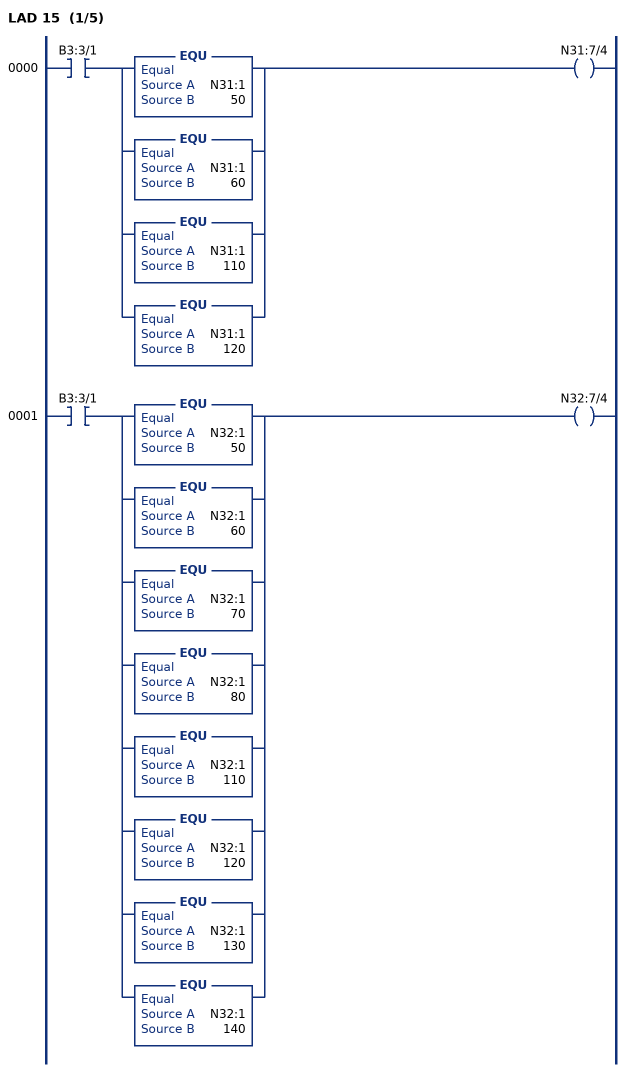
% Rung: 0 %
SOR XIC B3:3/1 BST EQU N31:1 50 NXB EQU N31:1 60 NXB EQU N31:1 110 NXB EQU N31:1 120 BND OTE N31:7/4 EOR
% Rung: 1 %
SOR XIC B3:3/1 BST EQU N32:1 50 NXB EQU N32:1 60 NXB EQU N32:1 70 NXB EQU N32:1 80 NXB EQU N32:1 110 NXB EQU N32:1 120 NXB EQU N32:1 130 NXB EQU N32:1 140 BND OTE N32:7/4 EOR

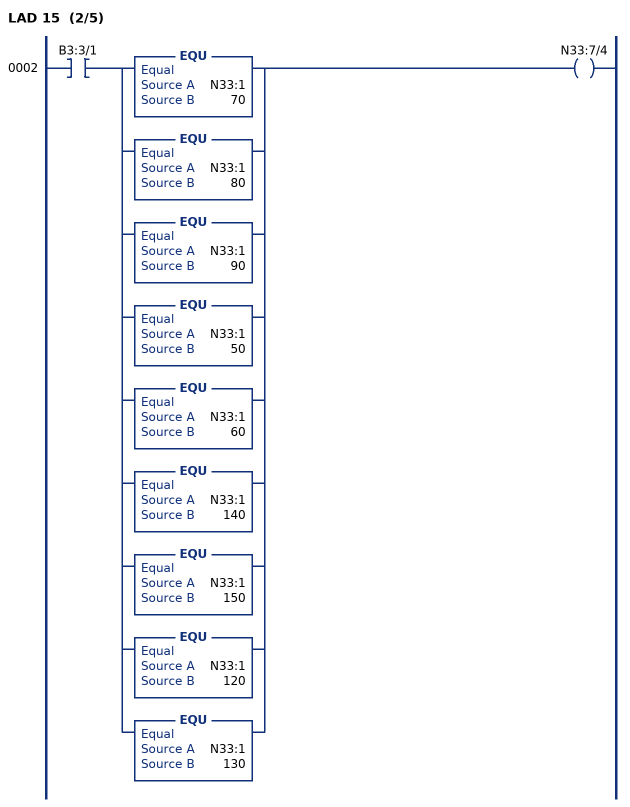
% Rung: 2 %
SOR XIC B3:3/1 BST EQU N33:1 70 NXB EQU N33:1 80 NXB EQU N33:1 90 NXB EQU N33:1 50 NXB EQU N33:1 60 NXB EQU N33:1 140 NXB EQU N33:1 150 NXB EQU N33:1 120 NXB EQU N33:1 130 BND OTE N33:7/4 EOR

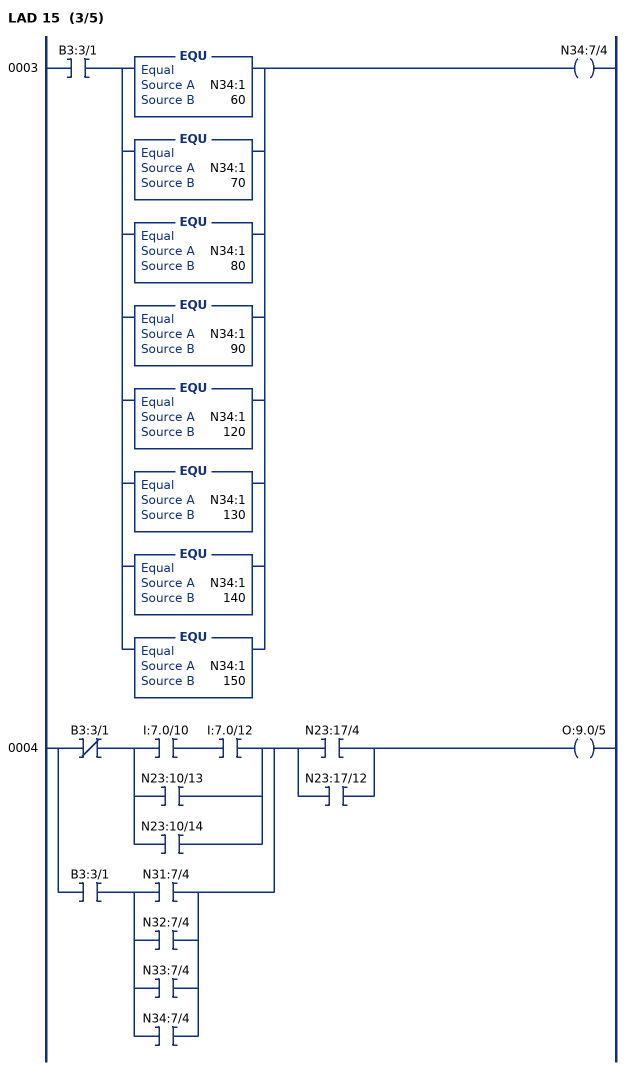
% Rung: 3 %
SOR XIC B3:3/1 BST EQU N34:1 60 NXB EQU N34:1 70 NXB EQU N34:1 80 NXB EQU N34:1 90 NXB EQU N34:1 120 NXB EQU N34:1 130 NXB EQU N34:1 140 NXB EQU N34:1 150 BND OTE N34:7/4 EOR
% Rung: 4 %
SOR BST XIO B3:3/1 BST XIC I:7.0/10 XIC I:7.0/12 NXB XIC N23:10/13 NXB XIC N23:10/14 BND NXB XIC B3:3/1 BST XIC N31:7/4 NXB XIC N32:7/4 NXB XIC N33:7/4 NXB XIC N34:7/4 BND BND BST XIC N23:17/4 NXB XIC N23:17/12 BND OTE O:9.0/5 EOR

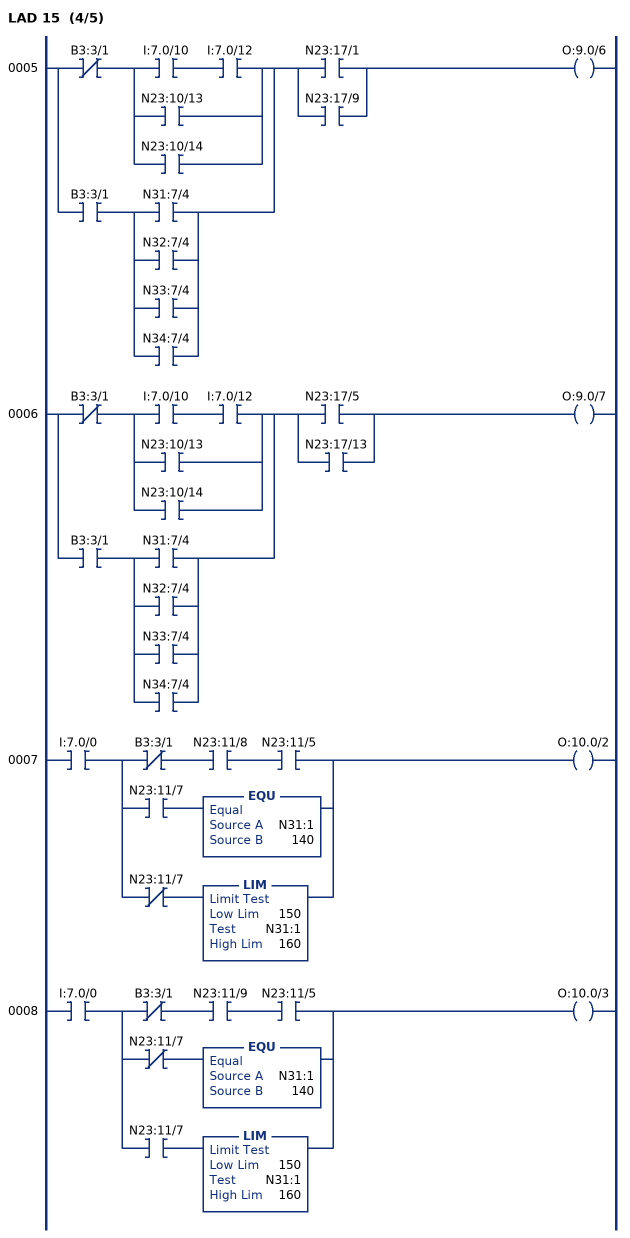
% Rung: 5 %
SOR BST XIO B3:3/1 BST XIC I:7.0/10 XIC I:7.0/12 NXB XIC N23:10/13 NXB XIC N23:10/14 BND NXB XIC B3:3/1 BST XIC N31:7/4 NXB XIC N32:7/4 NXB XIC N33:7/4 NXB XIC N34:7/4 BND BND BST XIC N23:17/1 NXB XIC N23:17/9 BND OTE O:9.0/6 EOR
% Rung: 6 %
SOR BST XIO B3:3/1 BST XIC I:7.0/10 XIC I:7.0/12 NXB XIC N23:10/13 NXB XIC N23:10/14 BND NXB XIC B3:3/1 BST XIC N31:7/4 NXB XIC N32:7/4 NXB XIC N33:7/4 NXB XIC N34:7/4 BND BND BST XIC N23:17/5 NXB XIC N23:17/13 BND OTE O:9.0/7 EOR
% Rung: 7 %
SOR XIC I:7.0/0 BST XIO B3:3/1 XIC N23:11/8 XIC N23:11/5 NXB XIC N23:11/7 EQU N31:1 140 NXB XIO N23:11/7 LIM 150 N31:1 160 BND OTE O:10.0/2 EOR
% Rung: 8 %
SOR XIC I:7.0/0 BST XIO B3:3/1 XIC N23:11/9 XIC N23:11/5 NXB XIO N23:11/7 EQU N31:1 140 NXB XIC N23:11/7 LIM 150 N31:1 160 BND OTE O:10.0/3 EOR

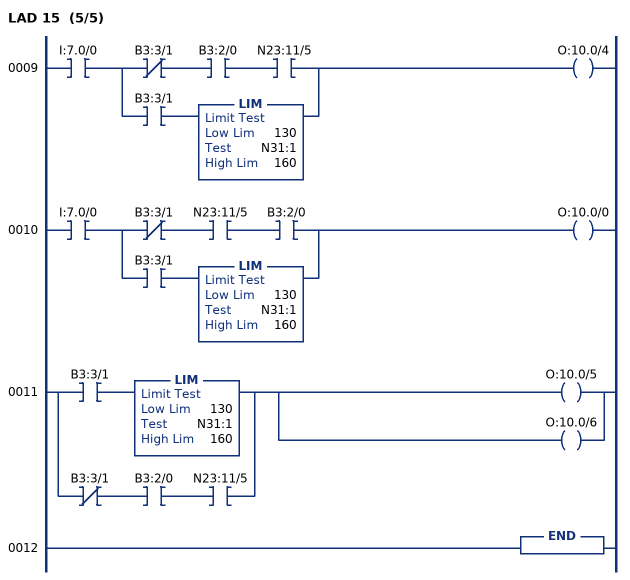
% Rung: 9 %
SOR XIC I:7.0/0 BST XIO B3:3/1 XIC B3:2/0 XIC N23:11/5 NXB XIC B3:3/1 LIM 130 N31:1 160 BND OTE O:10.0/4 EOR
% Rung: 10 %
SOR XIC I:7.0/0 BST XIO B3:3/1 XIC N23:11/5 XIC B3:2/0 NXB XIC B3:3/1 LIM 130 N31:1 160 BND OTE O:10.0/0 EOR
% Rung: 11 %
SOR BST XIC B3:3/1 LIM 130 N31:1 160 NXB XIO B3:3/1 XIC B3:2/0 XIC N23:11/5 BND BST OTE O:10.0/5 NXB OTE O:10.0/6 BND EOR
% Rung: 12 %
SOR END EOR

LADDER 21
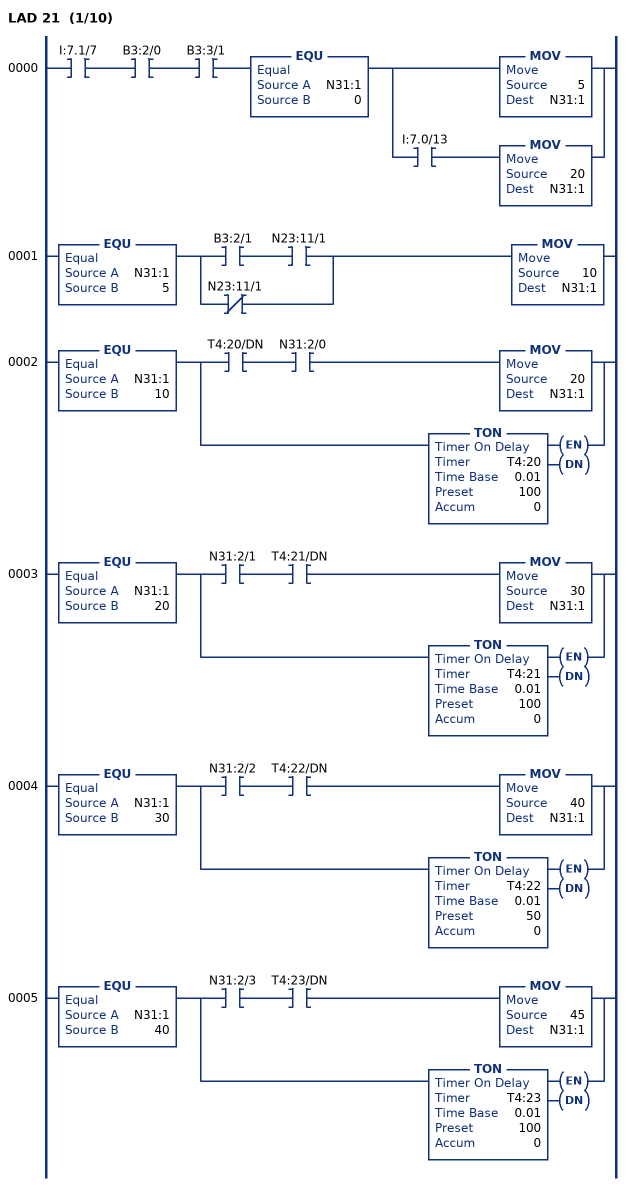
% Rung: 0 %
SOR XIC I:7.1/7 XIC B3:2/0 XIC B3:3/1 EQU N31:1 0 BST MOV 5 N31:1 NXB XIC I:7.0/13 MOV 20 N31:1 BND EOR
% Rung: 1 %
SOR EQU N31:1 5 BST XIC B3:2/1 XIC N23:11/1 NXB XIO N23:11/1 BND MOV 10 N31:1 EOR
% Rung: 2 %
SOR EQU N31:1 10 BST XIC T4:20/DN XIC N31:2/0 MOV 20 N31:1 NXB TON T4:20 0.01 100 0 BND EOR
% Rung: 3 %
SOR EQU N31:1 20 BST XIC N31:2/1 XIC T4:21/DN MOV 30 N31:1 NXB TON T4:21 0.01 100 0 BND EOR
% Rung: 4 %
SOR EQU N31:1 30 BST XIC N31:2/2 XIC T4:22/DN MOV 40 N31:1 NXB TON T4:22 0.01 50 0 BND EOR
% Rung: 5 %
SOR EQU N31:1 40 BST XIC N31:2/3 XIC T4:23/DN MOV 45 N31:1 NXB TON T4:23 0.01 100 0 BND EOR

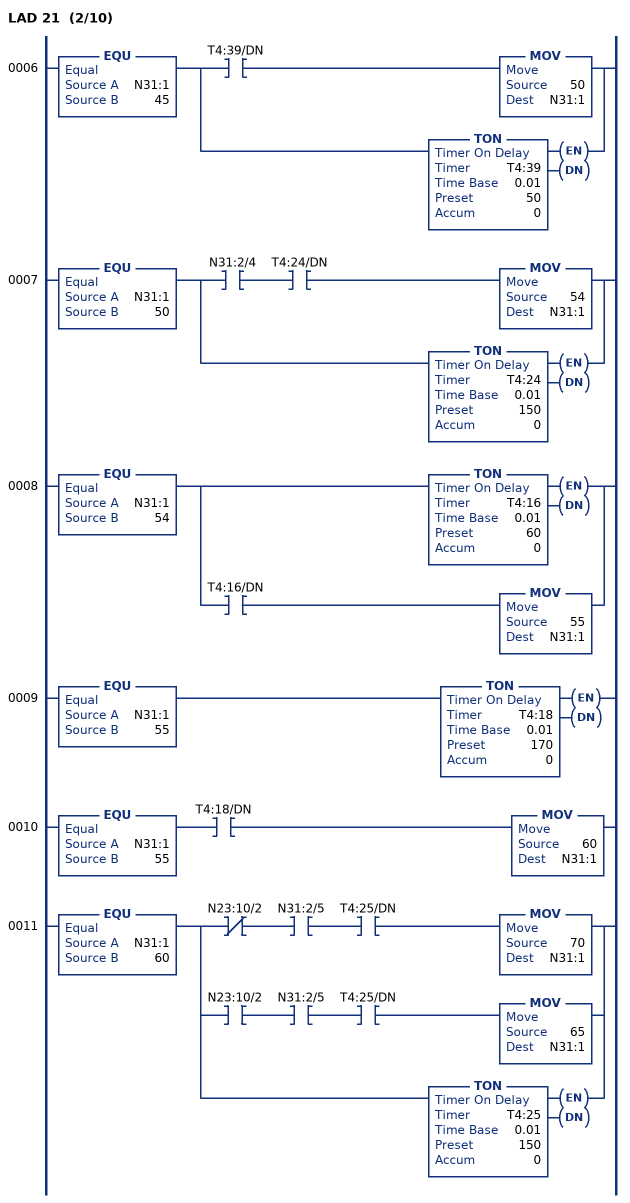
% Rung: 6 %
SOR EQU N31:1 45 BST XIC T4:39/DN MOV 50 N31:1 NXB TON T4:39 0.01 50 0 BND EOR
% Rung: 7 %
SOR EQU N31:1 50 BST XIC N31:2/4 XIC T4:24/DN MOV 54 N31:1 NXB TON T4:24 0.01 150 0 BND EOR
% Rung: 8 %
SOR EQU N31:1 54 BST TON T4:16 0.01 60 0 NXB XIC T4:16/DN MOV 55 N31:1 BND EOR
% Rung: 9 %
SOR EQU N31:1 55 TON T4:18 0.01 170 0 EOR
% Rung: 10 %
SOR EQU N31:1 55 XIC T4:18/DN MOV 60 N31:1 EOR
% Rung: 11 %
SOR EQU N31:1 60 BST XIO N23:10/2 XIC N31:2/5 XIC T4:25/DN MOV 70 N31:1 NXB XIC N23:10/2 XIC N31:2/5 XIC T4:25/DN MOV 65 N31:1 NXB TON T4:25 0.01 150 0 BND EOR

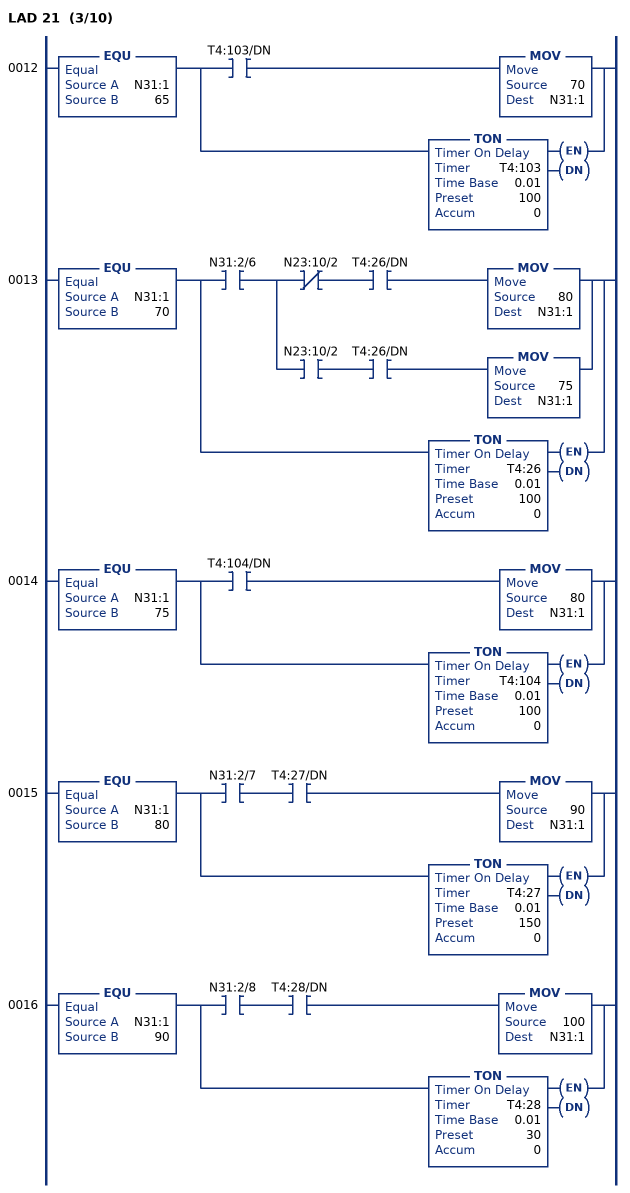
% Rung: 12 %
SOR EQU N31:1 65 BST XIC T4:103/DN MOV 70 N31:1 NXB TON T4:103 0.01 100 0 BND EOR
% Rung: 13 %
SOR EQU N31:1 70 BST XIC N31:2/6 BST XIO N23:10/2 XIC T4:26/DN MOV 80 N31:1 NXB XIC N23:10/2 XIC T4:26/DN MOV 75 N31:1 BND NXB TON T4:26 0.01 100 0 BND EOR
% Rung: 14 %
SOR EQU N31:1 75 BST XIC T4:104/DN MOV 80 N31:1 NXB TON T4:104 0.01 100 0 BND EOR
% Rung: 15 %
SOR EQU N31:1 80 BST XIC N31:2/7 XIC T4:27/DN MOV 90 N31:1 NXB TON T4:27 0.01 150 0 BND EOR
% Rung: 16 %
SOR EQU N31:1 90 BST XIC N31:2/8 XIC T4:28/DN MOV 100 N31:1 NXB TON T4:28 0.01 30 0 BND EOR

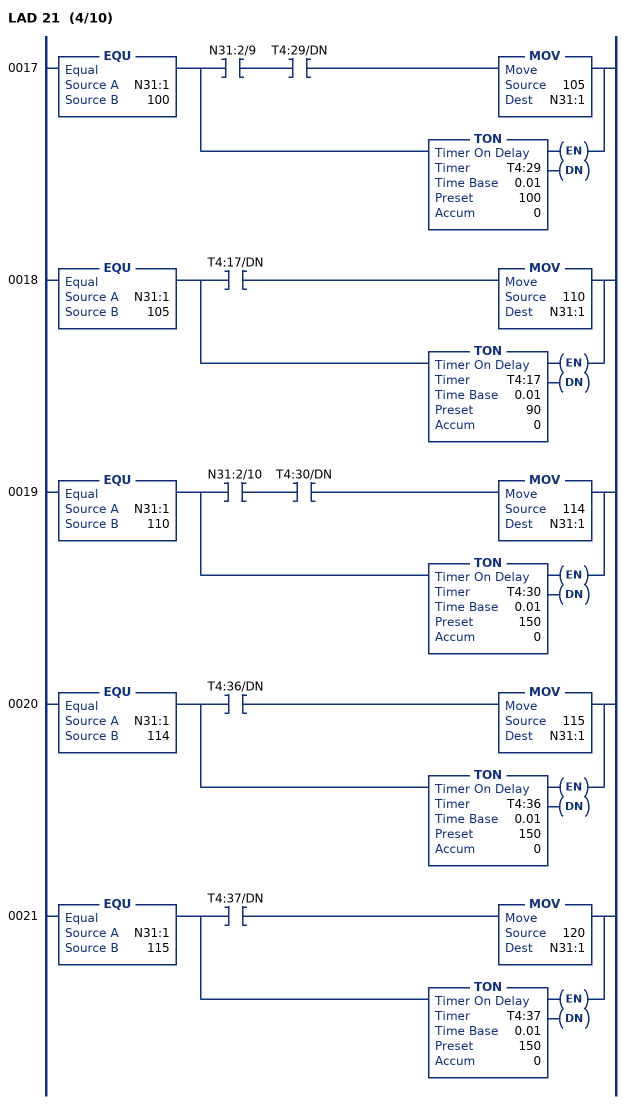
% Rung: 17 %
SOR EQU N31:1 100 BST XIC N31:2/9 XIC T4:29/DN MOV 105 N31:1 NXB TON T4:29 0.01 100 0 BND EOR
% Rung: 18 %
SOR EQU N31:1 105 BST XIC T4:17/DN MOV 110 N31:1 NXB TON T4:17 0.01 90 0 BND EOR
% Rung: 19 %
SOR EQU N31:1 110 BST XIC N31:2/10 XIC T4:30/DN MOV 114 N31:1 NXB TON T4:30 0.01 150 0 BND EOR
% Rung: 20 %
SOR EQU N31:1 114 BST XIC T4:36/DN MOV 115 N31:1 NXB TON T4:36 0.01 150 0 BND EOR
% Rung: 21 %
SOR EQU N31:1 115 BST XIC T4:37/DN MOV 120 N31:1 NXB TON T4:37 0.01 150 0 BND EOR

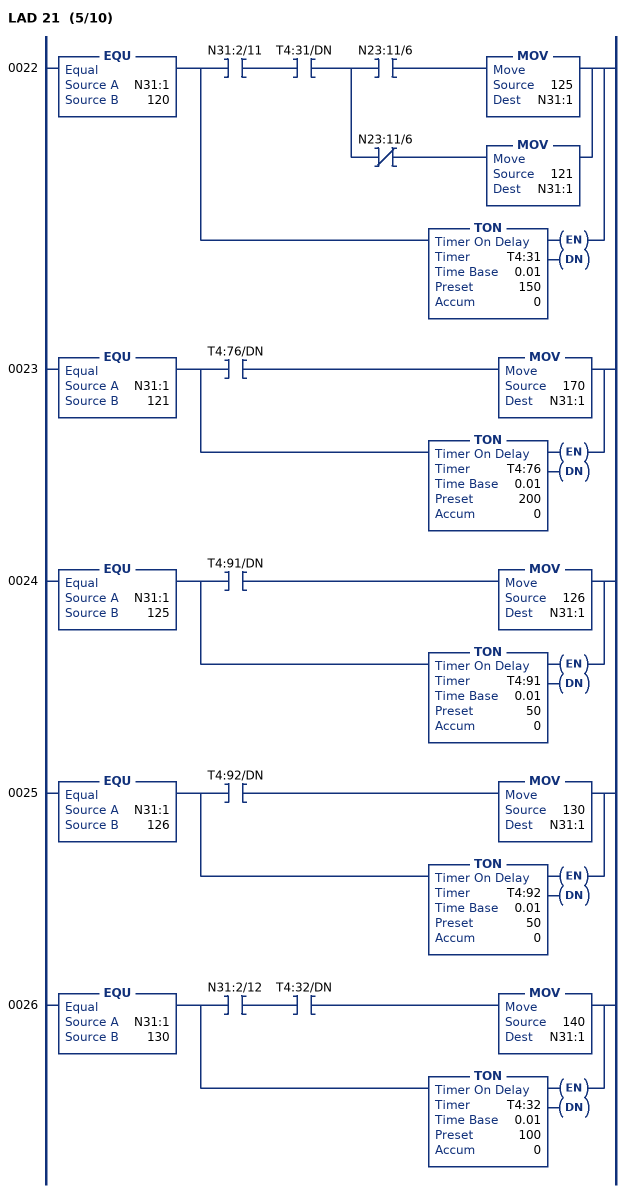
% Rung: 22 %
SOR EQU N31:1 120 BST XIC N31:2/11 XIC T4:31/DN BST XIC N23:11/6 MOV 125 N31:1 NXB XIO N23:11/6 MOV 121 N31:1 BND NXB TON T4:31 0.01 150 0 BND EOR
% Rung: 23 %
SOR EQU N31:1 121 BST XIC T4:76/DN MOV 170 N31:1 NXB TON T4:76 0.01 200 0 BND EOR
% Rung: 24 %
SOR EQU N31:1 125 BST XIC T4:91/DN MOV 126 N31:1 NXB TON T4:91 0.01 50 0 BND EOR
% Rung: 25 %
SOR EQU N31:1 126 BST XIC T4:92/DN MOV 130 N31:1 NXB TON T4:92 0.01 50 0 BND EOR
% Rung: 26 %
SOR EQU N31:1 130 BST XIC N31:2/12 XIC T4:32/DN MOV 140 N31:1 NXB TON T4:32 0.01 100 0 BND EOR

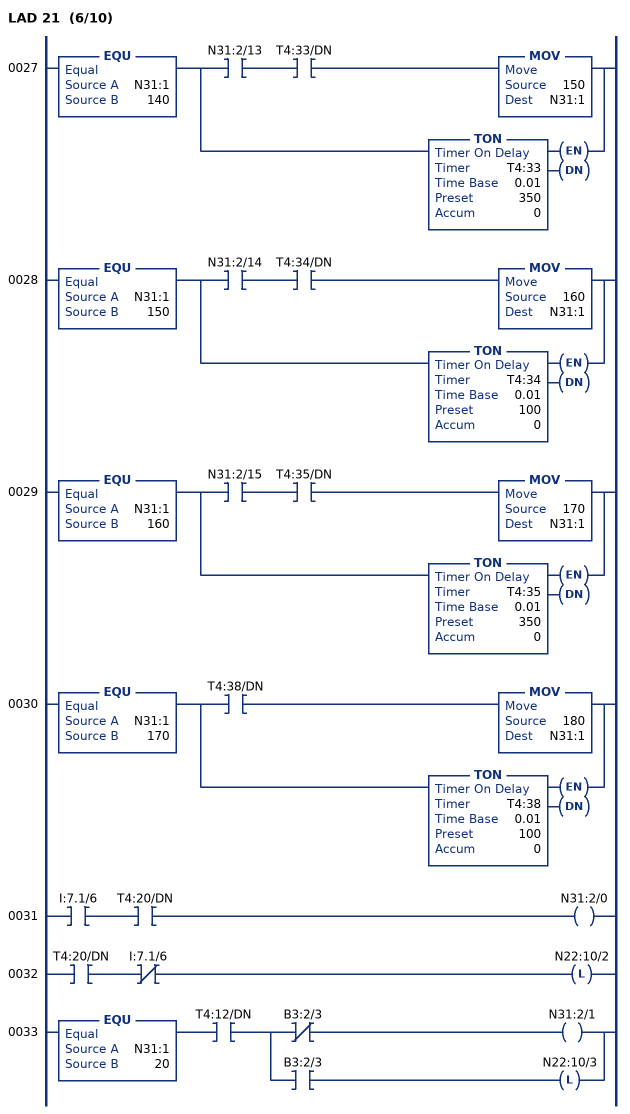
% Rung: 27 %
SOR EQU N31:1 140 BST XIC N31:2/13 XIC T4:33/DN MOV 150 N31:1 NXB TON T4:33 0.01 350 0 BND EOR
% Rung: 28 %
SOR EQU N31:1 150 BST XIC N31:2/14 XIC T4:34/DN MOV 160 N31:1 NXB TON T4:34 0.01 100 0 BND EOR
% Rung: 29 %
SOR EQU N31:1 160 BST XIC N31:2/15 XIC T4:35/DN MOV 170 N31:1 NXB TON T4:35 0.01 350 0 BND EOR
% Rung: 30 %
SOR EQU N31:1 170 BST XIC T4:38/DN MOV 180 N31:1 NXB TON T4:38 0.01 100 0 BND EOR
% Rung: 31 %
SOR XIC I:7.1/6 XIC T4:20/DN OTE N31:2/0 EOR
% Rung: 32 %
SOR XIC T4:20/DN XIO I:7.1/6 OTL N22:10/2 EOR
% Rung: 33 %
SOR EQU N31:1 20 XIC T4:12/DN BST XIO B3:2/3 OTE N31:2/1 NXB XIC B3:2/3 OTL N22:10/3 BND EOR

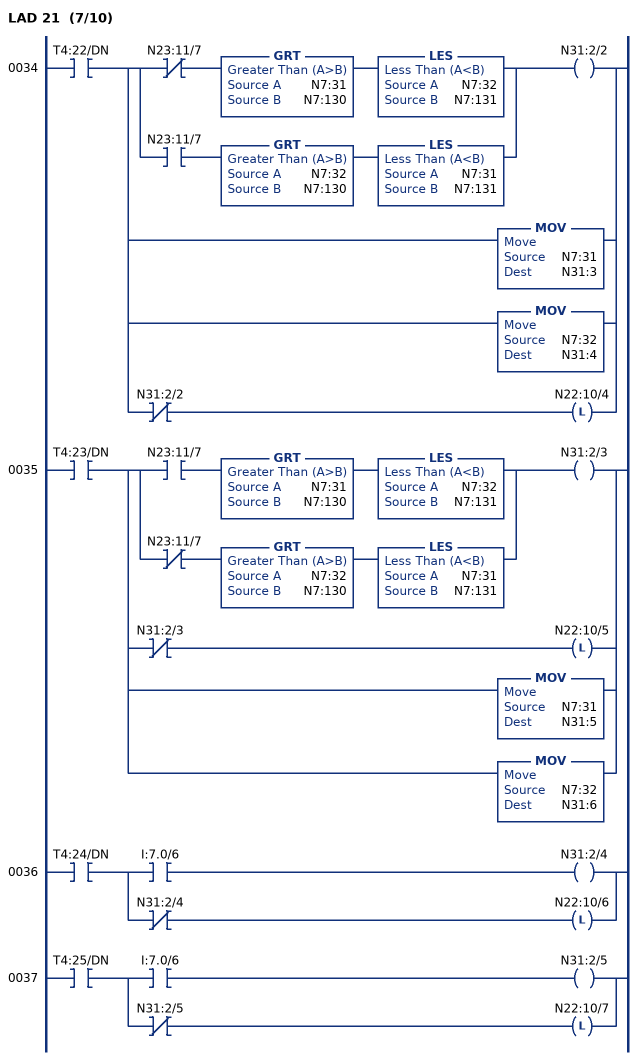
% Rung: 34 %
SOR XIC T4:22/DN BST BST XIO N23:11/7 GRT N7:31 N7:130 LES N7:32 N7:131 NXB XIC N23:11/7 GRT N7:32 N7:130 LES N7:31 N7:131 BND OTE N31:2/2 NXB BST MOV N7:31 N31:3 NXB MOV N7:32 N31:4 BND NXB XIO N31:2/2 OTL N22:10/4 BND EOR
% Rung: 35 %
SOR XIC T4:23/DN BST BST XIC N23:11/7 GRT N7:31 N7:130 LES N7:32 N7:131 NXB XIO N23:11/7 GRT N7:32 N7:130 LES N7:31 N7:131 BND OTE N31:2/3 NXB XIO N31:2/3 OTL N22:10/5 NXB BST MOV N7:31 N31:5 NXB MOV N7:32 N31:6 BND BND EOR
% Rung: 36 %
SOR XIC T4:24/DN BST XIC I:7.0/6 OTE N31:2/4 NXB XIO N31:2/4 OTL N22:10/6 BND EOR
% Rung: 37 %
SOR XIC T4:25/DN BST XIC I:7.0/6 OTE N31:2/5 NXB XIO N31:2/5 OTL N22:10/7 BND EOR

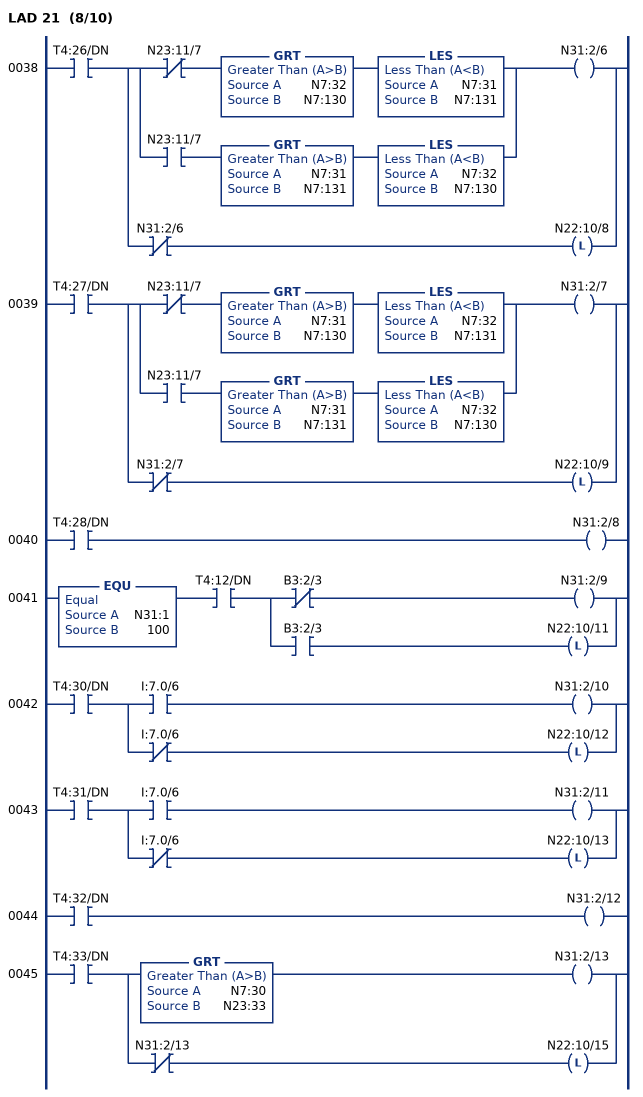
% Rung: 38 %
SOR XIC T4:26/DN BST BST XIO N23:11/7 GRT N7:32 N7:130 LES N7:31 N7:131 NXB XIC N23:11/7 GRT N7:31 N7:131 LES N7:32 N7:130 BND OTE N31:2/6 NXB XIO N31:2/6 OTL N22:10/8 BND EOR
% Rung: 39 %
SOR XIC T4:27/DN BST BST XIO N23:11/7 GRT N7:31 N7:130 LES N7:32 N7:131 NXB XIC N23:11/7 GRT N7:31 N7:131 LES N7:32 N7:130 BND OTE N31:2/7 NXB XIO N31:2/7 OTL N22:10/9 BND EOR
% Rung: 40 %
SOR XIC T4:28/DN OTE N31:2/8 EOR
% Rung: 41 %
SOR EQU N31:1 100 XIC T4:12/DN BST XIO B3:2/3 OTE N31:2/9 NXB XIC B3:2/3 OTL N22:10/11 BND EOR
% Rung: 42 %
SOR XIC T4:30/DN BST XIC I:7.0/6 OTE N31:2/10 NXB XIO I:7.0/6 OTL N22:10/12 BND EOR
% Rung: 43 %
SOR XIC T4:31/DN BST XIC I:7.0/6 OTE N31:2/11 NXB XIO I:7.0/6 OTL N22:10/13 BND EOR
% Rung: 44 %
SOR XIC T4:32/DN OTE N31:2/12 EOR
% Rung: 45 %
SOR XIC T4:33/DN BST GRT N7:30 N23:33 OTE N31:2/13 NXB XIO N31:2/13 OTL N22:10/15 BND EOR

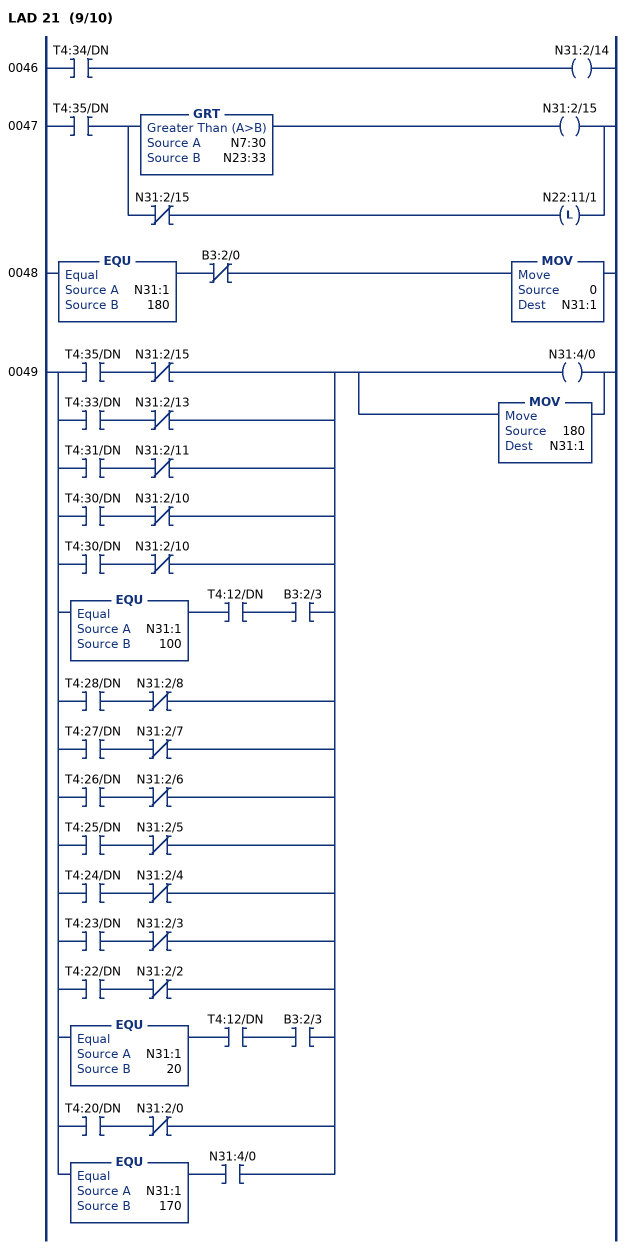
% Rung: 46 %
SOR XIC T4:34/DN OTE N31:2/14 EOR
% Rung: 47 %
SOR XIC T4:35/DN BST GRT N7:30 N23:33 OTE N31:2/15 NXB XIO N31:2/15 OTL N22:11/1 BND EOR
% Rung: 48 %
SOR EQU N31:1 180 XIO B3:2/0 MOV 0 N31:1 EOR
% Rung: 49 %
SOR BST XIC T4:35/DN XIO N31:2/15 NXB XIC T4:33/DN XIO N31:2/13 NXB XIC T4:31/DN XIO N31:2/11 NXB XIC T4:30/DN XIO N31:2/10 NXB XIC T4:30/DN XIO N31:2/10 NXB EQU N31:1 100 XIC T4:12/DN XIC B3:2/3 NXB XIC T4:28/DN XIO N31:2/8 NXB XIC T4:27/DN XIO N31:2/7 NXB XIC T4:26/DN XIO N31:2/6 NXB XIC T4:25/DN XIO N31:2/5 NXB XIC T4:24/DN XIO N31:2/4 NXB XIC T4:23/DN XIO N31:2/3 NXB XIC T4:22/DN XIO N31:2/2 NXB EQU N31:1 20 XIC T4:12/DN XIC B3:2/3 NXB XIC T4:20/DN XIO N31:2/0 NXB EQU N31:1 170 XIC N31:4/0 BND BST OTE N31:4/0 NXB MOV 180 N31:1 BND EOR

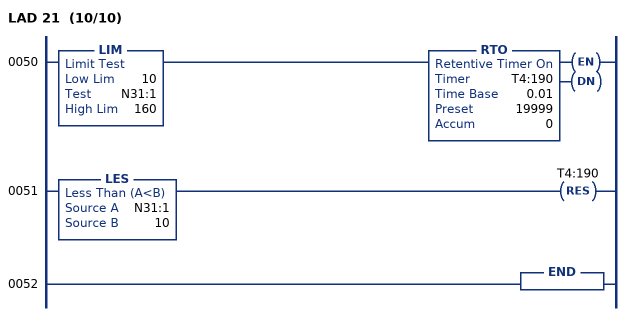
% Rung: 50 %
SOR LIM 10 N31:1 160 RTO T4:190 0.01 19999 0 EOR
% Rung: 51 %
SOR LES N31:1 10 RES T4:190 EOR
% Rung: 52 %
SOR END EOR

LADDER 22
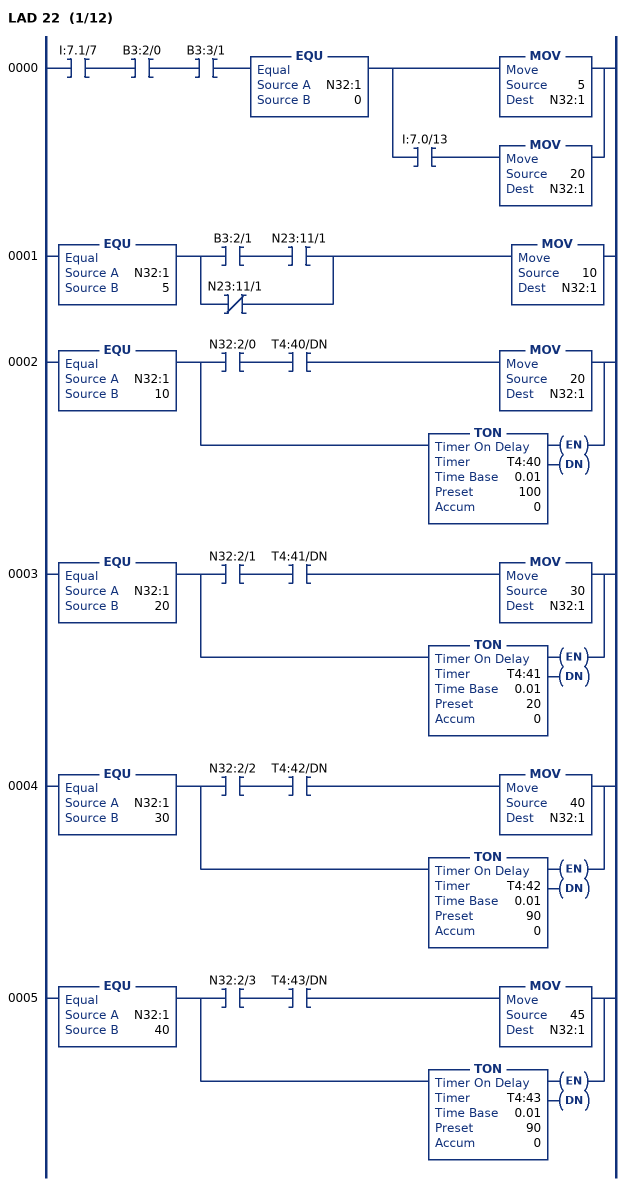
% Rung: 0 %
SOR XIC I:7.1/7 XIC B3:2/0 XIC B3:3/1 EQU N32:1 0 BST MOV 5 N32:1 NXB XIC I:7.0/13 MOV 20 N32:1 BND EOR
% Rung: 1 %
SOR EQU N32:1 5 BST XIC B3:2/1 XIC N23:11/1 NXB XIO N23:11/1 BND MOV 10 N32:1 EOR
% Rung: 2 %
SOR EQU N32:1 10 BST XIC N32:2/0 XIC T4:40/DN MOV 20 N32:1 NXB TON T4:40 0.01 100 0 BND EOR
% Rung: 3 %
SOR EQU N32:1 20 BST XIC N32:2/1 XIC T4:41/DN MOV 30 N32:1 NXB TON T4:41 0.01 20 0 BND EOR
% Rung: 4 %
SOR EQU N32:1 30 BST XIC N32:2/2 XIC T4:42/DN MOV 40 N32:1 NXB TON T4:42 0.01 90 0 BND EOR
% Rung: 5 %
SOR EQU N32:1 40 BST XIC N32:2/3 XIC T4:43/DN MOV 45 N32:1 NXB TON T4:43 0.01 90 0 BND EOR

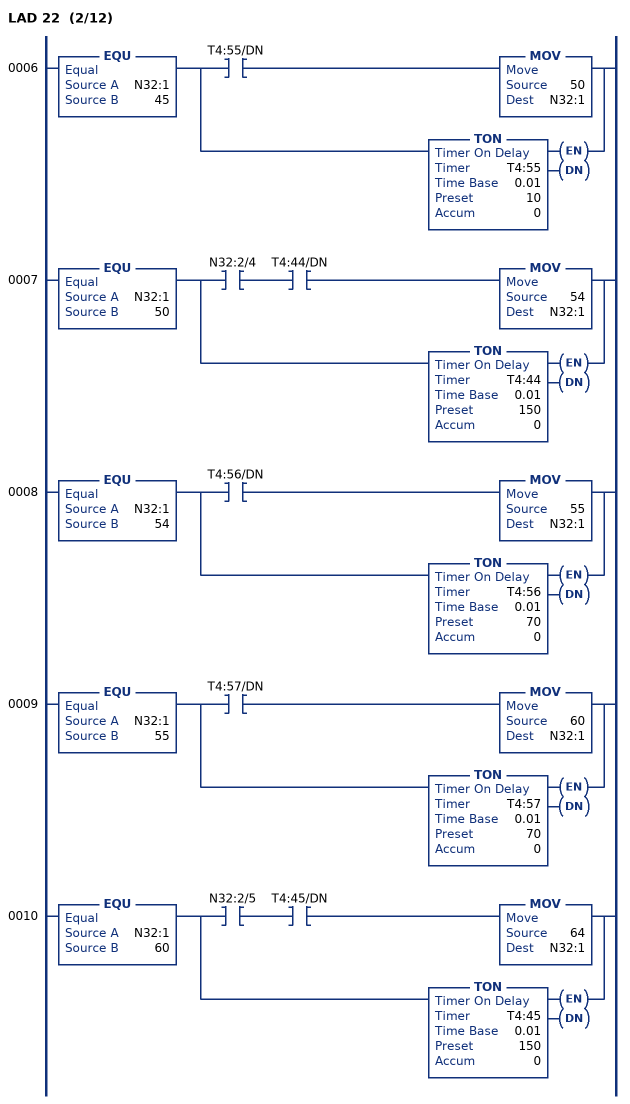
% Rung: 6 %
SOR EQU N32:1 45 BST XIC T4:55/DN MOV 50 N32:1 NXB TON T4:55 0.01 10 0 BND EOR
% Rung: 7 %
SOR EQU N32:1 50 BST XIC N32:2/4 XIC T4:44/DN MOV 54 N32:1 NXB TON T4:44 0.01 150 0 BND EOR
% Rung: 8 %
SOR EQU N32:1 54 BST XIC T4:56/DN MOV 55 N32:1 NXB TON T4:56 0.01 70 0 BND EOR
% Rung: 9 %
SOR EQU N32:1 55 BST XIC T4:57/DN MOV 60 N32:1 NXB TON T4:57 0.01 70 0 BND EOR
% Rung: 10 %
SOR EQU N32:1 60 BST XIC N32:2/5 XIC T4:45/DN MOV 64 N32:1 NXB TON T4:45 0.01 150 0 BND EOR

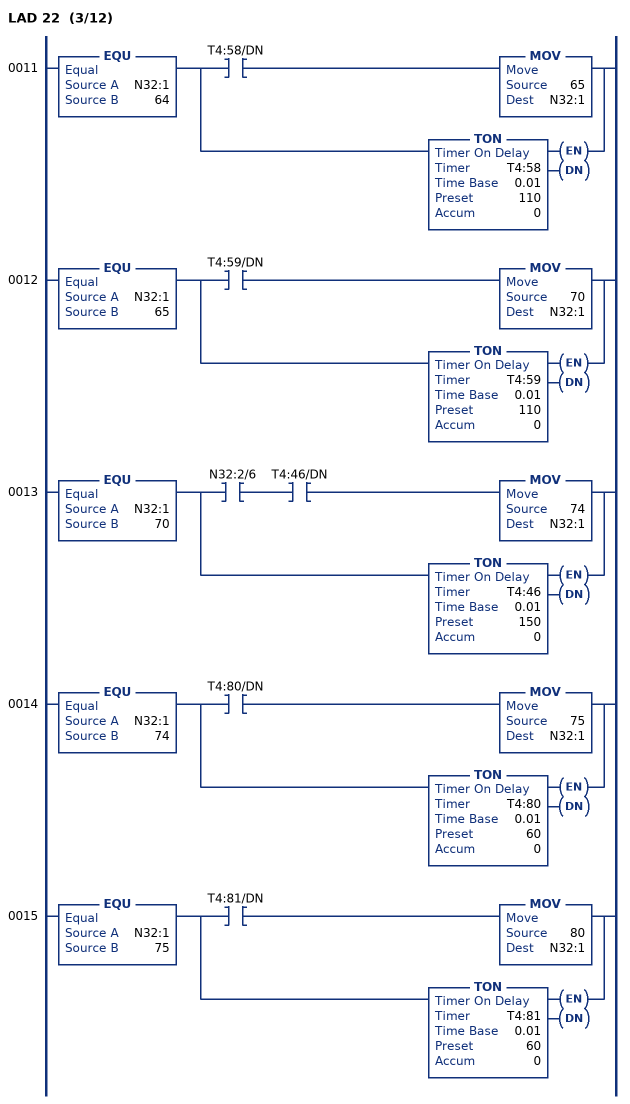
% Rung: 11 %
SOR EQU N32:1 64 BST XIC T4:58/DN MOV 65 N32:1 NXB TON T4:58 0.01 110 0 BND EOR
% Rung: 12 %
SOR EQU N32:1 65 BST XIC T4:59/DN MOV 70 N32:1 NXB TON T4:59 0.01 110 0 BND EOR
% Rung: 13 %
SOR EQU N32:1 70 BST XIC N32:2/6 XIC T4:46/DN MOV 74 N32:1 NXB TON T4:46 0.01 150 0 BND EOR
% Rung: 14 %
SOR EQU N32:1 74 BST XIC T4:80/DN MOV 75 N32:1 NXB TON T4:80 0.01 60 0 BND EOR
% Rung: 15 %
SOR EQU N32:1 75 BST XIC T4:81/DN MOV 80 N32:1 NXB TON T4:81 0.01 60 0 BND EOR

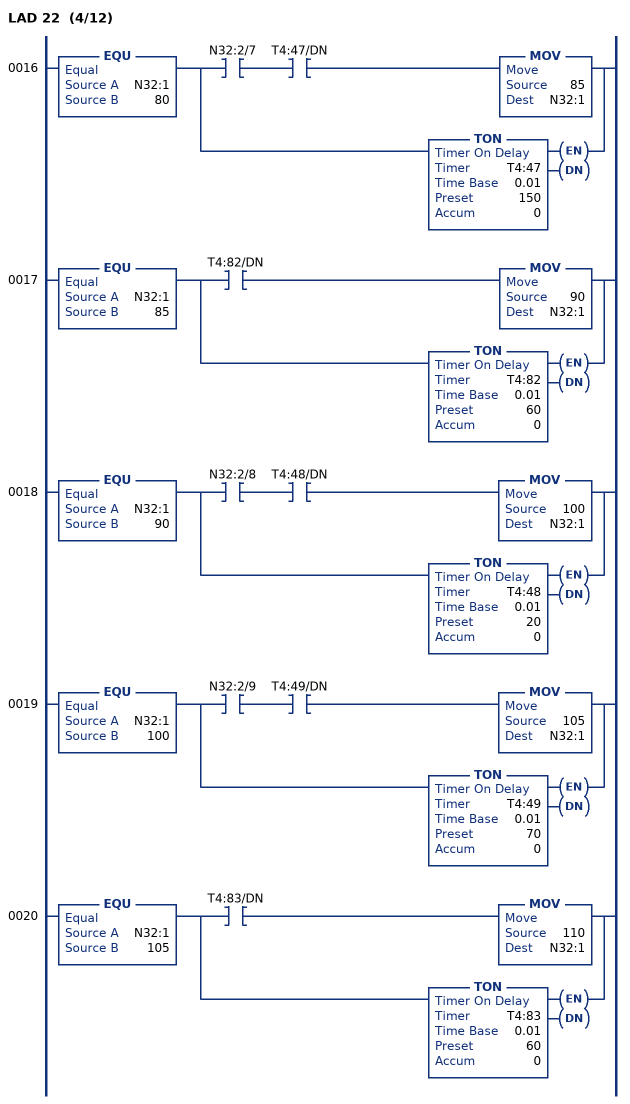
% Rung: 16 %
SOR EQU N32:1 80 BST XIC N32:2/7 XIC T4:47/DN MOV 85 N32:1 NXB TON T4:47 0.01 150 0 BND EOR
% Rung: 17 %
SOR EQU N32:1 85 BST XIC T4:82/DN MOV 90 N32:1 NXB TON T4:82 0.01 60 0 BND EOR
% Rung: 18 %
SOR EQU N32:1 90 BST XIC N32:2/8 XIC T4:48/DN MOV 100 N32:1 NXB TON T4:48 0.01 20 0 BND EOR
% Rung: 19 %
SOR EQU N32:1 100 BST XIC N32:2/9 XIC T4:49/DN MOV 105 N32:1 NXB TON T4:49 0.01 70 0 BND EOR
% Rung: 20 %
SOR EQU N32:1 105 BST XIC T4:83/DN MOV 110 N32:1 NXB TON T4:83 0.01 60 0 BND EOR

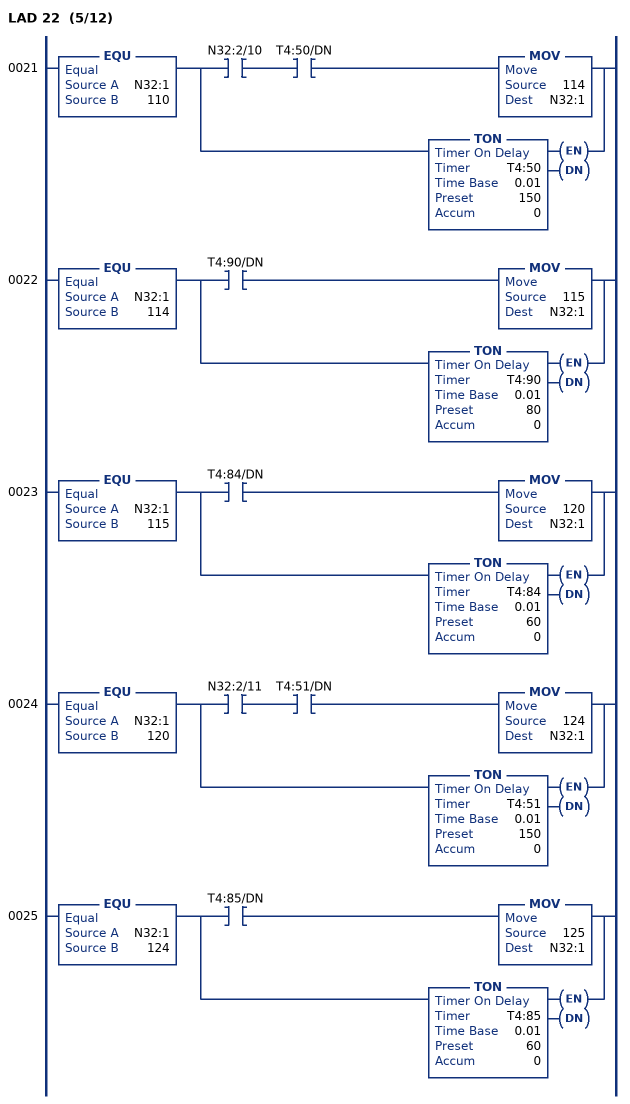
% Rung: 21 %
SOR EQU N32:1 110 BST XIC N32:2/10 XIC T4:50/DN MOV 114 N32:1 NXB TON T4:50 0.01 150 0 BND EOR
% Rung: 22 %
SOR EQU N32:1 114 BST XIC T4:90/DN MOV 115 N32:1 NXB TON T4:90 0.01 80 0 BND EOR
% Rung: 23 %
SOR EQU N32:1 115 BST XIC T4:84/DN MOV 120 N32:1 NXB TON T4:84 0.01 60 0 BND EOR
% Rung: 24 %
SOR EQU N32:1 120 BST XIC N32:2/11 XIC T4:51/DN MOV 124 N32:1 NXB TON T4:51 0.01 150 0 BND EOR
% Rung: 25 %
SOR EQU N32:1 124 BST XIC T4:85/DN MOV 125 N32:1 NXB TON T4:85 0.01 60 0 BND EOR

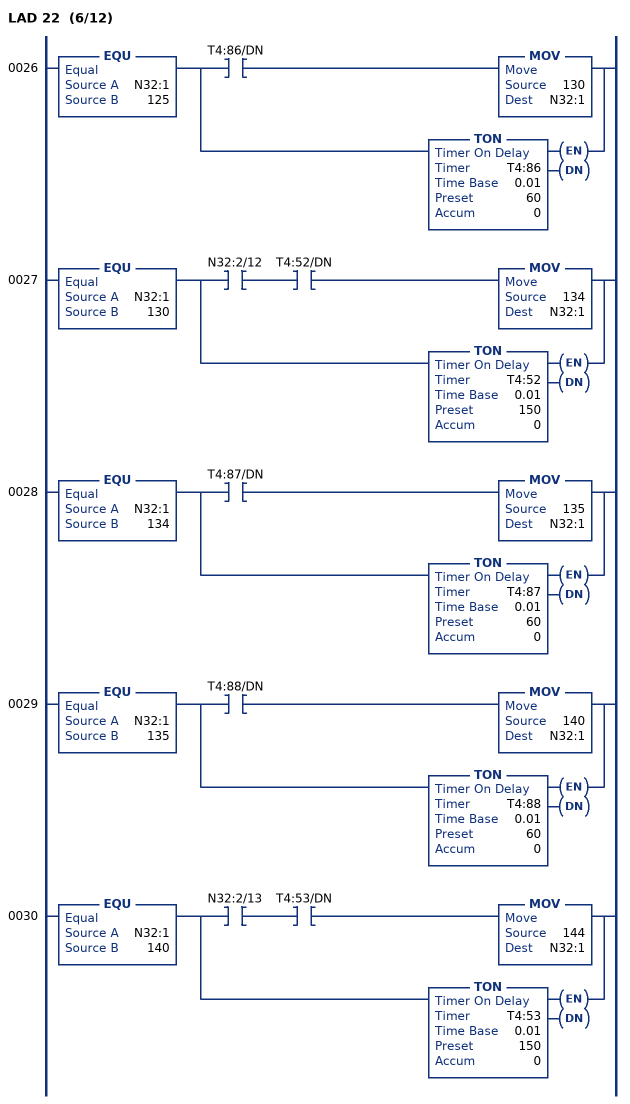
% Rung: 26 %
SOR EQU N32:1 125 BST XIC T4:86/DN MOV 130 N32:1 NXB TON T4:86 0.01 60 0 BND EOR
% Rung: 27 %
SOR EQU N32:1 130 BST XIC N32:2/12 XIC T4:52/DN MOV 134 N32:1 NXB TON T4:52 0.01 150 0 BND EOR
% Rung: 28 %
SOR EQU N32:1 134 BST XIC T4:87/DN MOV 135 N32:1 NXB TON T4:87 0.01 60 0 BND EOR
% Rung: 29 %
SOR EQU N32:1 135 BST XIC T4:88/DN MOV 140 N32:1 NXB TON T4:88 0.01 60 0 BND EOR
% Rung: 30 %
SOR EQU N32:1 140 BST XIC N32:2/13 XIC T4:53/DN MOV 144 N32:1 NXB TON T4:53 0.01 150 0 BND EOR

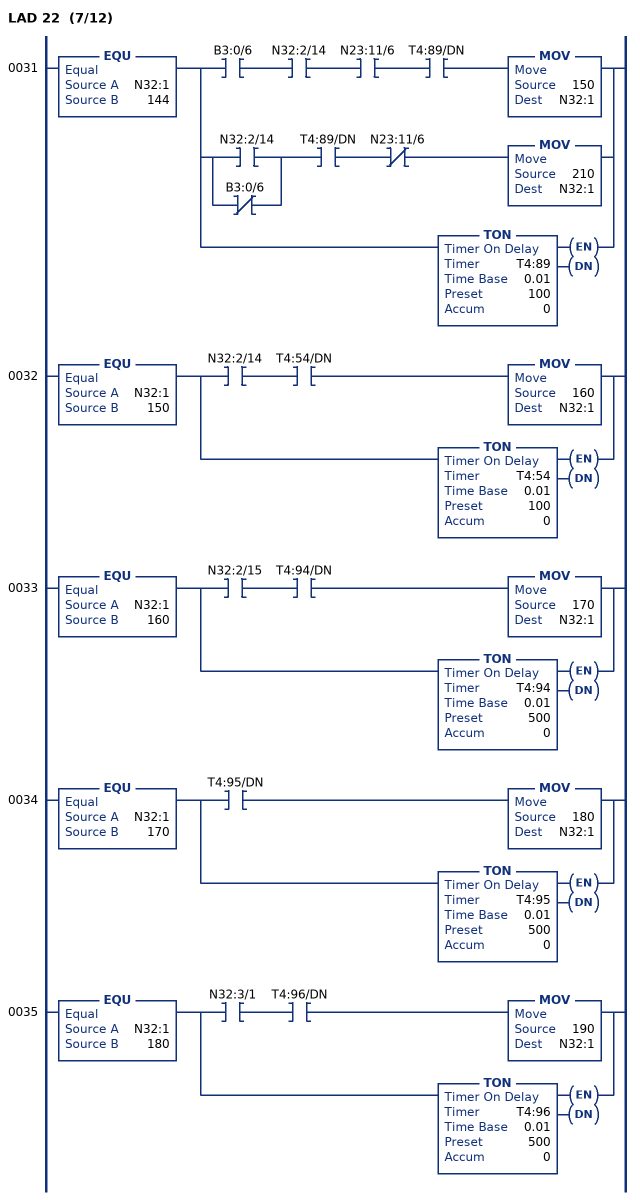
% Rung: 31 %
SOR EQU N32:1 144 BST XIC B3:0/6 XIC N32:2/14 XIC N23:11/6 XIC T4:89/DN MOV 150 N32:1 NXB BST XIC N32:2/14 NXB XIO B3:0/6 BND XIC T4:89/DN XIO N23:11/6 MOV 210 N32:1 NXB TON T4:89 0.01 100 0 BND EOR
% Rung: 32 %
SOR EQU N32:1 150 BST XIC N32:2/14 XIC T4:54/DN MOV 160 N32:1 NXB TON T4:54 0.01 100 0 BND EOR
% Rung: 33 %
SOR EQU N32:1 160 BST XIC N32:2/15 XIC T4:94/DN MOV 170 N32:1 NXB TON T4:94 0.01 500 0 BND EOR
% Rung: 34 %
SOR EQU N32:1 170 BST XIC T4:95/DN MOV 180 N32:1 NXB TON T4:95 0.01 500 0 BND EOR
% Rung: 35 %
SOR EQU N32:1 180 BST XIC N32:3/1 XIC T4:96/DN MOV 190 N32:1 NXB TON T4:96 0.01 500 0 BND EOR

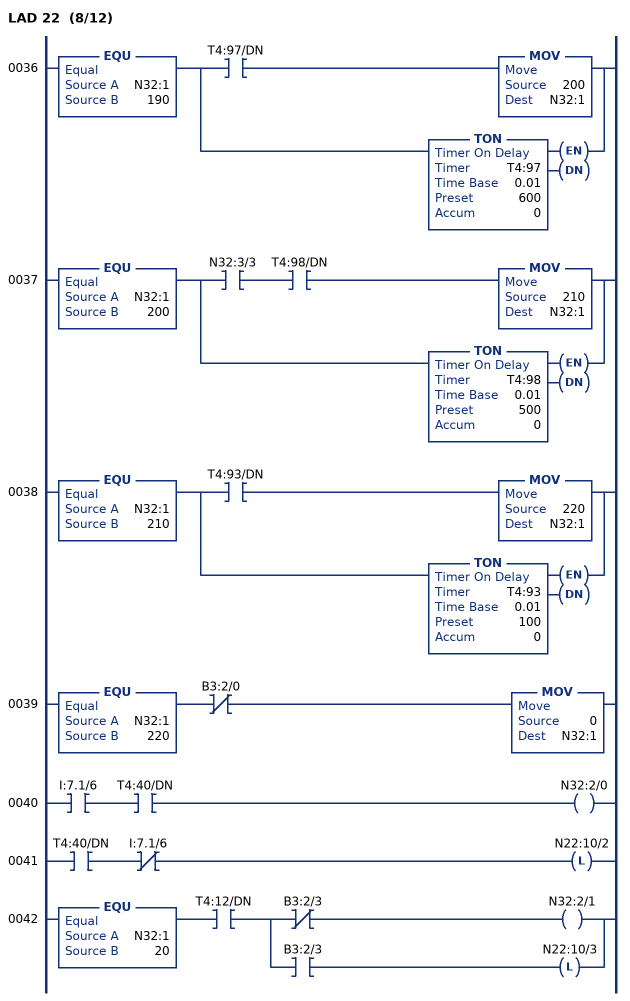
% Rung: 36 %
SOR EQU N32:1 190 BST XIC T4:97/DN MOV 200 N32:1 NXB TON T4:97 0.01 600 0 BND EOR
% Rung: 37 %
SOR EQU N32:1 200 BST XIC N32:3/3 XIC T4:98/DN MOV 210 N32:1 NXB TON T4:98 0.01 500 0 BND EOR
% Rung: 38 %
SOR EQU N32:1 210 BST XIC T4:93/DN MOV 220 N32:1 NXB TON T4:93 0.01 100 0 BND EOR
% Rung: 39 %
SOR EQU N32:1 220 XIO B3:2/0 MOV 0 N32:1 EOR
% Rung: 40 %
SOR XIC I:7.1/6 XIC T4:40/DN OTE N32:2/0 EOR
% Rung: 41 %
SOR XIC T4:40/DN XIO I:7.1/6 OTL N22:10/2 EOR
% Rung: 42 %
SOR EQU N32:1 20 XIC T4:12/DN BST XIO B3:2/3 OTE N32:2/1 NXB XIC B3:2/3 OTL N22:10/3 BND EOR

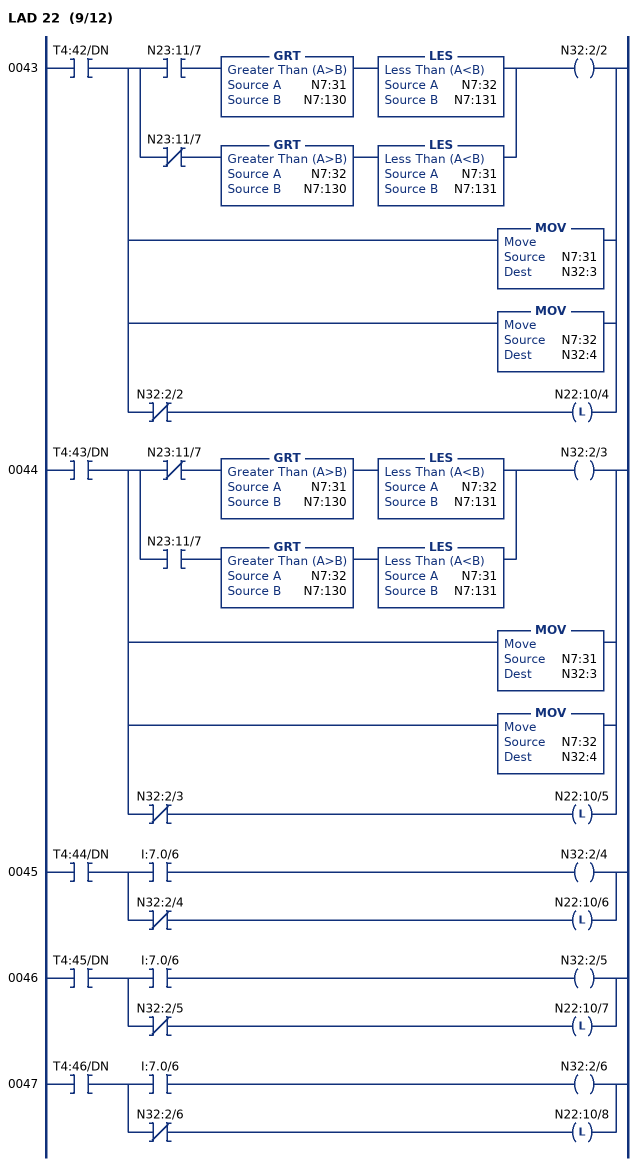
% Rung: 43 %
SOR XIC T4:42/DN BST BST XIC N23:11/7 GRT N7:31 N7:130 LES N7:32 N7:131 NXB XIO N23:11/7 GRT N7:32 N7:130 LES N7:31 N7:131 BND OTE N32:2/2 NXB BST MOV N7:31 N32:3 NXB MOV N7:32 N32:4 BND NXB XIO N32:2/2 OTL N22:10/4 BND EOR
% Rung: 44 %
SOR XIC T4:43/DN BST BST XIO N23:11/7 GRT N7:31 N7:130 LES N7:32 N7:131 NXB XIC N23:11/7 GRT N7:32 N7:130 LES N7:31 N7:131 BND OTE N32:2/3 NXB BST MOV N7:31 N32:3 NXB MOV N7:32 N32:4 BND NXB XIO N32:2/3 OTL N22:10/5 BND EOR
% Rung: 45 %
SOR XIC T4:44/DN BST XIC I:7.0/6 OTE N32:2/4 NXB XIO N32:2/4 OTL N22:10/6 BND EOR
% Rung: 46 %
SOR XIC T4:45/DN BST XIC I:7.0/6 OTE N32:2/5 NXB XIO N32:2/5 OTL N22:10/7 BND EOR
% Rung: 47 %
SOR XIC T4:46/DN BST XIC I:7.0/6 OTE N32:2/6 NXB XIO N32:2/6 OTL N22:10/8 BND EOR

